ADAPTER ATimeTick (* Interface for a time out service roughly based on the definitions of ROOM *)
  (* Standard: 61499-1; Description: Copyright (c) 2017 fortiss GmbH This program and the accompanying materials are made available under the terms of the Eclipse Public License 2.0 which is available at https://www.eclipse.org/legal/epl-2.0/ SPDX-License-Identifier: EPL-2.0 *)
  (* Version 3.1, 2026-08-14, Franz Höpfinger, HR Agrartechnik GmbH, FB_TON like cyclic Interface *)
  (* Version 3.0, 2025-04-14, Patrick Aigner, changed package *)
  (* Version 1.0, 2017-09-22, Alois Zoitl, fortiss GmbH, initial API and implementation and/or initial documentation *)
  PACKAGE adapter::events::TimeOut;
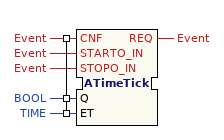
  EVENT_INPUT
    CNF WITH Q, ET; (* Execution Confirmation *)
    STARTO_IN;
    STOPO_IN;
  END_EVENT
  EVENT_OUTPUT
    REQ; (* Normal Execution Request *)
  END_EVENT
  VAR_INPUT
    Q : BOOL; (* is started = TRUE *)
    ET : TIME; (* Elapsed time *)
  END_VAR
  SERVICE SOCKET/PLUG
    SEQUENCE Timeout
      PLUG.START(TD) -> SOCKET.START(TD);
      SOCKET.TimeOut() -> PLUG.TimeOut();
    END_SEQUENCE
    SEQUENCE NormalOperation
      PLUG.Start(TD) -> SOCKET.Start(TD);
      PLUG.STOP() -> SOCKET.STOP();
    END_SEQUENCE
  END_SERVICE
END_ADAPTER
